// TIA Portal V17 export
// export: Created 2023-05-07T12:12:21.7473379Z, ExportSetting WithDefaults, DisplayName Totally Integrated Automation Portal, DisplayVersion V17, DisplayName TIA Portal Openness, DisplayVersion V17, DisplayName TIA Portal Version Control Interface, DisplayVersion V17, DisplayName TIA Portal Test Suite Advanced, DisplayVersion V17, DisplayName STEP 7 Professional, DisplayVersion V17, DisplayName SIMATIC Energy Suite, DisplayVersion V17, DisplayName STEP 7 Safety, DisplayVersion V17, DisplayName WinCC Professional, DisplayVersion V17
FUNCTION "VisuClass" : Void   // FC8, LAD
TITLE = VisuClass
{ S7_Optimized_Access := 'TRUE' }
VERSION : 0.1
// stored: AutoNumber true, IsIECCheckEnabled false, SetENOAutomatically false, UDAEnableTagReadback false
BEGIN

REGION Network 1: Call: StartStop
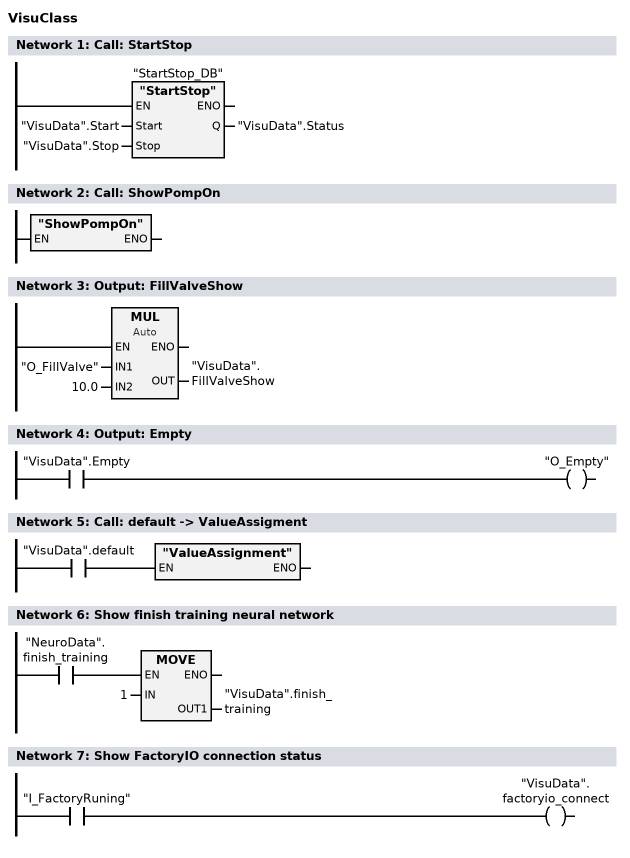
   RUNG wire#powerrail
      "StartStop_DB"(Start := "VisuData".Start, Stop := "VisuData".Stop, Q => "VisuData".Status)
   END_RUNG
   // the same network as SCL:
   "StartStop_DB"(Start := "VisuData".Start, Stop := "VisuData".Stop, Q => "VisuData".Status);   // "StartStop"
END_REGION

REGION Network 2: Call: ShowPompOn
   RUNG wire#powerrail
      "ShowPompOn"()
   END_RUNG
   // the same network as SCL:
   "ShowPompOn"();
END_REGION

REGION Network 3: Output: FillValveShow
   RUNG wire#powerrail
      Mul(in1 := "O_FillValve", in2 := 10.0, out => "VisuData".FillValveShow)
   END_RUNG
   // the same network as SCL:
   "VisuData".FillValveShow := "O_FillValve" * 10.0;
END_REGION

REGION Network 4: Output: Empty
   RUNG wire#powerrail
      Contact( "VisuData".Empty )
      Coil( "O_Empty" )
   END_RUNG
   // the same network as SCL:
   "O_Empty" := "VisuData".Empty;
END_REGION

REGION Network 5: Call: default -> ValueAssigment
   RUNG wire#powerrail
      Contact( "VisuData".default )
      "ValueAssignment"()
   END_RUNG
   // the same network as SCL:
   IF "VisuData".default THEN "ValueAssignment"(); END_IF;
END_REGION

REGION Network 6: Show finish training neural network
   RUNG wire#powerrail
      Contact( "NeuroData".finish_training )
      Move(in := 1, out1 => "VisuData".finish_training)
   END_RUNG
   // the same network as SCL:
   IF "NeuroData".finish_training THEN "VisuData".finish_training := 1; END_IF;
END_REGION

REGION Network 7: Show FactoryIO connection status
   RUNG wire#powerrail
      Contact( "I_FactoryRuning" )
      Coil( "VisuData".factoryio_connect )
   END_RUNG
   // the same network as SCL:
   "VisuData".factoryio_connect := "I_FactoryRuning";
END_REGION
END_FUNCTION
